// TIA Portal V20 export
TYPE "Temperature_DT"
   STRUCT
      axFactor : Real := 1.0;
      bOffset : Real := 0.0;
   END_STRUCT;
END_TYPE
